FUNCTION "GetBitByte" : Bool   // FC2, SCL
{ S7_Optimized_Access := 'TRUE' }
VERSION : 0.1
   VAR_INPUT
      Data : Byte;
      pos : Int;
   END_VAR
   VAR_TEMP
      mask : Byte;
      temp : Byte;
   END_VAR
BEGIN
   #mask := 1;
   IF #pos < 8 THEN
       #mask := SHL(IN := #mask, N := #pos);
       #temp := #Data AND #mask;
       #GetBitByte := (#temp > 0);
   ELSE
       #GetBitByte := 0;
   END_IF;
END_FUNCTION

FUNCTION "GetBitWord" : Bool   // FC3, SCL
{ S7_Optimized_Access := 'TRUE' }
VERSION : 0.1
   VAR_INPUT
      Data : Word;
      pos : Int;
   END_VAR
   VAR_TEMP
      mask : Word;
      temp : Word;
   END_VAR
BEGIN
   #mask := 1;
   IF #pos < 16 THEN
       #mask := SHL(IN := #mask, N := #pos);
       #temp := #Data AND #mask;
       #GetBitWord := (#temp > 0);
   ELSE
       #GetBitWord := 0;
   END_IF;
END_FUNCTION

FUNCTION "SwapWord" : Void   // FC4, SCL
{ S7_Optimized_Access := 'TRUE' }
VERSION : 0.1
   VAR_INPUT
      NDB : Int;   // Номер DB-источника данных
      offset : Int;   // Смещение от начала DB, в байтах
      "counter" : Int;   // Число переворачиваемых WORD-ов
   END_VAR
   VAR_TEMP
      peek1 : Byte;
      peek2 : Byte;
      i : Int;
   END_VAR
BEGIN

   FOR #i := #offset TO #offset + (#counter - 1) * 2 BY 2 DO
       #peek1 := PEEK(area := 16#84,
                      dbNumber := #NDB,
                      byteOffset := #i);
       #peek2 := PEEK(area := 16#84,
                      dbNumber := #NDB,
                      byteOffset := #i + 1);
       POKE(area := 16#84,
            dbNumber := #NDB,
            byteOffset := #i + 1,
            value := #peek1);
       POKE(area := 16#84,
            dbNumber := #NDB,
            byteOffset := #i,
            value := #peek2);
   END_FOR;
END_FUNCTION

FUNCTION "Swap_float" : Void   // FC5, SCL
{ S7_Optimized_Access := 'TRUE' }
VERSION : 0.1
   VAR_INPUT
      offset : Int;
      "counter" : Int;
      NDB : Int;
   END_VAR
   VAR_TEMP
      i : Int;
      peek1 : Word;
      peek2 : Word;
   END_VAR
BEGIN
   FOR #i := #offset TO #offset + (#counter - 1) * 4 BY 4 DO
       #peek1 := PEEK_WORD(area := 16#84,
                           dbNumber := #NDB,
                           byteOffset := #i);
       #peek2 := PEEK_WORD(area := 16#84,
                           dbNumber := #NDB,
                           byteOffset := #i + 2);
       POKE(area := 16#84,
            dbNumber := #NDB,
            byteOffset := #i + 2,
            value := #peek1);
       POKE(area := 16#84,
            dbNumber := #NDB,
            byteOffset := #i,
            value := #peek2);
   END_FOR;
END_FUNCTION

FUNCTION "SetBitWord" : Void   // FC6, SCL
{ S7_Optimized_Access := 'TRUE' }
VERSION : 0.1
   VAR_INPUT
      pos : Int;
      value : Bool;
   END_VAR
   VAR_IN_OUT
      Data : Word;
   END_VAR
   VAR_TEMP
      mask : Word;
      v : Word;
   END_VAR
BEGIN
   IF #pos < 16 THEN
       #mask := 1;
       #mask := SHL(IN := #mask, N := #pos);
       IF #value THEN
           #Data := #Data OR #mask;
       ELSE
           #Data := #Data AND (NOT #mask);
       END_IF;
   END_IF;
END_FUNCTION

FUNCTION "SetBitByte" : Void   // FC7, SCL
{ S7_Optimized_Access := 'TRUE' }
VERSION : 0.1
   VAR_INPUT
      pos : Int;
      value : Bool;
   END_VAR
   VAR_IN_OUT
      Data : Byte;
   END_VAR
   VAR_TEMP
      mask : Byte;
      v : Byte;
   END_VAR
BEGIN
   IF #pos < 8 THEN
       #mask := 1;
       #mask := SHL(IN := #mask, N := #pos);
       IF #value THEN
           #Data := #Data OR #mask;
       ELSE
           #Data := #Data AND (NOT #mask);
       END_IF;
   END_IF;
END_FUNCTION

// folder: Modbus

FUNCTION "UVP_Processing" : Void   // FC9, SCL
{ S7_Optimized_Access := 'TRUE' }
VERSION : 0.1
   VAR_TEMP
      NewState : Int;
      Cant_connect1 : Bool;
      Cant_connect2 : Bool;
      Cant_connect_with_UVP : Bool;
      Request_Finished : Bool;
      Request_Finished_with_Error : Bool;
      len : UInt;
   END_VAR
BEGIN
   // Установить IP адрес УВП
   (*IF "UVP_Data".Commands.Set_IP_UVP1 THEN
       IF NOT "UVP_States".Client.Disconnect THEN
           "UVP_States".Connect_UVP.ID := UINT_TO_WORD("UVP_Data".UVP1_Settings.Connect_ID);
           "UVP_States".Connect_UVP.RemoteAddress.ADDR[1] := UINT_TO_BYTE("UVP_Data".UVP1_Settings.IP_OCTET1);
           "UVP_States".Connect_UVP.RemoteAddress.ADDR[2] := UINT_TO_BYTE("UVP_Data".UVP1_Settings.IP_OCTET2);
           "UVP_States".Connect_UVP.RemoteAddress.ADDR[3] := UINT_TO_BYTE("UVP_Data".UVP1_Settings.IP_OCTET3);
           "UVP_States".Connect_UVP.RemoteAddress.ADDR[4] := UINT_TO_BYTE("UVP_Data".UVP1_Settings.IP_OCTET4);
           "UVP_States".Connect_UVP.RemotePort := "UVP_Data".UVP1_Settings.IP_PORT;
           "UVP_States".State := 10;
           "UVP_States".Client.Disconnect := True;
       ELSE
           "UVP_States".Client.Disconnect := False;
           "UVP_Data".Commands.Set_IP_UVP1 := False;
       END_IF;
   END_IF;*)

   #NewState := -1;

   // определение проблем с подключением
   #Request_Finished := "UVP_States".Client.Done OR "UVP_States".Client.Error OR ("UVP_States".Client.Busy AND ("UVP_States".Client.Status = 16#7002));
   // признак завершения цикла работы чтения/записи с ошибкой
   #Request_Finished_with_Error := ("UVP_States".Client.Busy AND ("UVP_States".Client.Status = 16#7002)) OR
   ("UVP_States".Client.Error AND (("UVP_States".Client.Status <> 16#7002)));

   // определение проблем со связью
   IF ("UVP_States".Client.Busy OR "UVP_States".Client.Error) THEN
       "UVP_off".TON (IN := true, PT := t#5s);
       IF "UVP_off".Q THEN
           "UVP_Data".Flags.UVP1_on := false;
           "ReqUVP" := 0;
           #NewState := "UVP_States".ReqReadOpData_nextState;
           "UVP_off".TON (IN := false, PT := t#5s);
       END_IF;
   ELSE
       "UVP_off".TON (IN := false, PT := t#5s);
   END_IF;

   IF "UVP_States".Client.Done AND (NOT "UVP_States".Client.Error) THEN
       "UVP_Data".Flags.UVP1_on := true;
   END_IF;

   (*IF "ReqUVP" THEN
       "ReqUVP" := 0;
   ELSE
       IF NOT ("UVP_States".Client.Done OR "UVP_States".Client.Error OR "UVP_States".Client.Busy) THEN
           "ReqUVP" := 1;
       END_IF;
   END_IF;*)


   CASE "UVP_States".State OF
       10..29:// State=10 - чтение оперативных данных первой линии, параметры с 3 по 23
           // State=11 - чтение накопленных данных первой линии, 4 группы по 5 параметров
           // State=12 - чтение оперативных данных первой линии, параметры с 1 по 3
           // 
           // State=13 - чтение оперативных данных второй линии, параметры с 3 по 23
           // State=14 - чтение накопленных данных второй линии, 4 группы по 5 параметров
           // State=15 - чтение оперативных данных второй линии, параметры с 1 по 3

           // 
           IF ("PrevState" <> "UVP_States".State) THEN
               "UVP_States".ReqReadOpData.Mode := 0;
               //ил 1
               IF "UVP_States".State = 10 THEN
                   "UVP_States".ReqReadOpData.Data_ADDR := 32001;
                   "UVP_States".ReqReadOpData.Data_LEN := 46;
                   "UVP_States".ReqReadOpData_dest_offset := 64; // смещение проверить в Дата
                   "UVP_States".ReqReadOpData_nextState := 11;
               ELSIF "UVP_States".State = 11 THEN
                   "UVP_States".ReqReadOpData.Data_ADDR := 32061;
                   "UVP_States".ReqReadOpData.Data_LEN := 40;
                   "UVP_States".ReqReadOpData_dest_offset := 156; // смещение проверить в Дата
                   "UVP_States".ReqReadOpData_nextState := 13;

                   //ил 2    
               ELSIF "UVP_States".State = 13 THEN
                   "UVP_States".ReqReadOpData.Data_ADDR := 32101;
                   "UVP_States".ReqReadOpData.Data_LEN := 46;
                   "UVP_States".ReqReadOpData_dest_offset := 236;
                   "UVP_States".ReqReadOpData_nextState := 14;
               ELSIF "UVP_States".State = 14 THEN
                   "UVP_States".ReqReadOpData.Data_ADDR := 32161;
                   "UVP_States".ReqReadOpData.Data_LEN := 40;
                   "UVP_States".ReqReadOpData_dest_offset := 328;
                   "UVP_States".ReqReadOpData_nextState := 30;
               END_IF;
               "ReqUVP" := 0;
               "UVP_States".ClientMode := "UVP_States".ReqReadOpData;
               "ReqUVP" := 1;

           END_IF;
           // обработка принятых данных
           IF "UVP_States".Client.Done THEN
               // перекладываем прочитаные данные в секцию UVP_Current_L1(L2), UVP_Current_L1(L2)  или UVP_Cumulative_L1(L3), смотря по запросу              
               "CopyWord"(NDBsrc := 14,
                          NDBdest := 13,
                          offset_src := 52,
                          offset_dest := "UVP_States".ReqReadOpData_dest_offset,
                          counter := UINT_TO_INT("UVP_States".ReqReadOpData.Data_LEN));
               "ReqUVP" := 0;
               // постобработка данных - перевожу Па в МПа, секундные расходы в часовые
               IF "UVP_States".State = 10 THEN
                   "UVP_Data".UVP1_Current_L1.UVP_mass_flow := "UVP_Data".UVP1_Current_L1.UVP_mass_flow * 3600.0;
                   "UVP_Data".UVP1_Current_L1.UVP_Param_m_flow := "UVP_Data".UVP1_Current_L1.UVP_Param_m_flow * 3600.0;
                   "UVP_Data".UVP1_Current_L1.UVP_Param_vol_flow_norm := "UVP_Data".UVP1_Current_L1.UVP_Param_vol_flow_norm * 3600.0;
                   "UVP_Data".UVP1_Current_L1.UVP_Param_vol_flow_work := "UVP_Data".UVP1_Current_L1.UVP_Param_vol_flow_work * 3600.0;
                   "UVP_Data".UVP1_Current_L1.UVP_vol_flow_norm := "UVP_Data".UVP1_Current_L1.UVP_vol_flow_norm * 3600.0;
                   "UVP_Data".UVP1_Current_L1.UVP_vol_flow_work := "UVP_Data".UVP1_Current_L1.UVP_vol_flow_work * 3600.0;
                   "UVP_Data".UVP1_Current_L1.UVP_Abs_press := "UVP_Data".UVP1_Current_L1.UVP_Abs_press / 1000000;
                   "UVP_Data".UVP1_Current_L1.UVP_Press := "UVP_Data".UVP1_Current_L1.UVP_Press / 1000000;
               ELSIF "UVP_States".State = 11 THEN
                   "UVP_Data".UVP1_Cumulative_L1.UVP_Mass_prev2h := "UVP_Data".UVP1_Cumulative_L1.UVP_Mass_prev2h / 1000.0;
                   "UVP_Data".UVP1_Cumulative_L1.UVP_Param_m_flow_prev2h := "UVP_Data".UVP1_Cumulative_L1.UVP_Param_m_flow_prev2h / 1000.0;
                   "UVP_Data".UVP1_Cumulative_L1.UVP_Mass_prevDay := "UVP_Data".UVP1_Cumulative_L1.UVP_Mass_prevDay / 1000.0;
                   "UVP_Data".UVP1_Cumulative_L1.UVP_Param_m_flow_prevDay := "UVP_Data".UVP1_Cumulative_L1.UVP_Param_m_flow_prevDay / 1000.0;
               ELSIF "UVP_States".State = 13 THEN
                   "UVP_Data".UVP1_Current_L2.UVP_mass_flow := "UVP_Data".UVP1_Current_L2.UVP_mass_flow * 3.6;
                   "UVP_Data".UVP1_Current_L2.UVP_Param_m_flow := "UVP_Data".UVP1_Current_L2.UVP_Param_m_flow * 3600.0;
                   "UVP_Data".UVP1_Current_L2.UVP_Param_vol_flow_norm := "UVP_Data".UVP1_Current_L2.UVP_Param_vol_flow_norm * 3600.0;
                   "UVP_Data".UVP1_Current_L2.UVP_Param_vol_flow_work := "UVP_Data".UVP1_Current_L2.UVP_Param_vol_flow_work * 3600.0;
                   "UVP_Data".UVP1_Current_L2.UVP_vol_flow_norm := "UVP_Data".UVP1_Current_L2.UVP_vol_flow_norm * 3600.0;
                   "UVP_Data".UVP1_Current_L2.UVP_vol_flow_work := "UVP_Data".UVP1_Current_L2.UVP_vol_flow_work * 3600.0;
                   "UVP_Data".UVP1_Current_L2.UVP_Abs_press := "UVP_Data".UVP1_Current_L2.UVP_Abs_press / 1000000;
                   "UVP_Data".UVP1_Current_L2.UVP_Press := "UVP_Data".UVP1_Current_L2.UVP_Press / 1000000;
               ELSIF "UVP_States".State = 14 THEN
                   "UVP_Data".UVP1_Cumulative_L2.UVP_Mass_prev2h := "UVP_Data".UVP1_Cumulative_L2.UVP_Mass_prev2h / 1000.0;
                   "UVP_Data".UVP1_Cumulative_L2.UVP_Param_m_flow_prev2h := "UVP_Data".UVP1_Cumulative_L2.UVP_Param_m_flow_prev2h / 1000.0;
                   "UVP_Data".UVP1_Cumulative_L2.UVP_Mass_prevDay := "UVP_Data".UVP1_Cumulative_L2.UVP_Mass_prevDay / 1000.0;
                   "UVP_Data".UVP1_Cumulative_L2.UVP_Param_m_flow_prevDay := "UVP_Data".UVP1_Cumulative_L2.UVP_Param_m_flow_prevDay / 1000.0;
               END_IF;
               // Переходим к следующему запросу
               #NewState := "UVP_States".ReqReadOpData_nextState;
           ELSIF #Request_Finished_with_Error THEN
               // Если не получается связаться - переходим к следующему запросу и продолжаем попытки
               #NewState := "UVP_States".ReqReadOpData_nextState;
           ELSE
               ;
           END_IF;

           //******************** проверка команд*************************************************************************************************

           IF "UVP_Data".Commands.UVPArchReadStart THEN
               // переход к чтению архивной записи
               #NewState := 55;
               //ELSIF "UVP_Data".Commands.UVP_MR113_Read THEN         //читаем циклически
               // переход к чтению компонентного состава газа
               //    #NewState := 40;
           ELSIF "UVP_Data".Commands.UVP_MR113_Write THEN
               // переход к записи компонентного состава газа
               #NewState := 50;

           ELSE
               // нет команды
               ;
           END_IF;

       30:  //  чтение часов реального времени выбранного УВП, сразу после измеряемых параметров УВП по обоим линиям         
           IF NOT "UVP_States".Client.Busy THEN
               "UVP_States".ReqReadOpData.Mode := 0;
               "UVP_States".ReqReadOpData.Data_ADDR := 41801;
               "UVP_States".ReqReadOpData.Data_LEN := 6;
               "ReqUVP" := 0;
               "UVP_States".ClientMode := "UVP_States".ReqReadOpData;
               "ReqUVP" := 1;
               #NewState := 31;
           END_IF;

       31: // обработка принятых данных часов реального времени выбранного УВП
           // крутить их не нужно, так как в УВП они в нормальном представлении
           IF "UVP_States".Client.Done THEN
               // перекладываем прочитаные данные в секцию UVP_DateTime
               "CopyWord"(NDBsrc := 14,
                          NDBdest := 13,
                          offset_src := 52,
                          offset_dest := 924,
                          counter := 6);
               "ReqUVP" := 0;
               #NewState := 32;
           ELSIF #Request_Finished_with_Error THEN
               // Если не получается связаться - переходим к следующему запросу и продолжаем попытки
               #NewState := 32;
           ELSE
               ;
           END_IF;

       32:  //  запись нужного порядка байт в 4-х байтной переменной         
           IF NOT "UVP_States".Client.Busy THEN
               "UVP_States".ReqWriteCom.Mode := 1;
               "UVP_States".ReqWriteCom.Data_ADDR := 40101;
               "UVP_States".ReqWriteCom.Data_LEN := 1;
               "ReqUVP" := 0;
               %DB14.DBW52 := 291;                                  // это 0123h
               "UVP_States".ClientMode := "UVP_States".ReqWriteCom;
               "ReqUVP" := 1;
               #NewState := 33;
           END_IF;

       33: // ожидание завершения записи порядка байт
           IF #Request_Finished THEN
               // Возвращаемся к очередному запросу (с которого нас сняли командой)
               #NewState := 40;
               "ReqUVP" := 0;
           END_IF;


       40:  // State=40 - запуск чтения компонентного состава газа
           IF NOT "UVP_States".Client.Busy THEN
               "UVP_States".ReqReadOpData.Mode := 0;
               "UVP_States".ReqReadOpData.Data_ADDR := 41103;
               "UVP_States".ReqReadOpData.Data_LEN := 30;
               "ReqUVP" := 0;
               "UVP_States".ClientMode := "UVP_States".ReqReadOpData;
               "ReqUVP" := 1;
               #NewState := 41;
           END_IF;

       41: // State=41 - обработка принятых данных компонентного состава газа
           IF "UVP_States".Client.Done THEN
               // перекладываем прочитаные данные в секцию UVP_MR113
               "CopyWord"(NDBsrc := 14,
                          NDBdest := 13,
                          offset_src := 52,
                          offset_dest := 936,
                          counter := 30);
               "ReqUVP" := 0;
               // Возвращаемся к очередному запросу (с которого нас сняли командой)
               #NewState := 42;
               "UVP_Data".Commands.UVP_MR113_Read := False;
           ELSIF #Request_Finished_with_Error THEN
               // Если не получается связаться - переходим к следующему запросу и продолжаем попытки
               #NewState := 42;
               //"UVP_v2_Data".Commands.UVP_MR113_Read := False; // Из-за этого не читает комп. состав при загрузке контроллера
           ELSE
               ;
           END_IF;


       42:  // State=42 - запуск чтения параметров: молярная или массовая концентрация,  влажность
           IF NOT "UVP_States".Client.Busy THEN
               "UVP_States".ReqReadOpData.Mode := 0;
               "UVP_States".ReqReadOpData.Data_ADDR := 41101;
               "UVP_States".ReqReadOpData.Data_LEN := 2;
               "ReqUVP" := 0;
               "UVP_States".ClientMode := "UVP_States".ReqReadOpData;
               "ReqUVP" := 1;
               #NewState := 43;
           END_IF;

       43: // State=43 - обработка принятых параметров: молярная или массовая концентрация,  влажность
           IF "UVP_States".Client.Done THEN
               // перекладываем прочитаные данные в секцию UVP_MR113
               // крутить их не нужно, так как в УВП они в нормальном представлении
               "CopyWord"(NDBsrc := 14,
                          NDBdest := 13,
                          offset_src := 52,
                          offset_dest := 996,
                          counter := 2);
               "ReqUVP" := 0;
               // Возвращаемся к очередному запросу (с которого нас сняли командой)
               #NewState := 10;
           ELSIF #Request_Finished_with_Error THEN
               // Если не получается связаться - переходим к следующему запросу и продолжаем попытки
               #NewState := 10;
           ELSE
               ;
           END_IF;// конец            

       50:  // State=50 - запись компонентного состава газа
           IF NOT "UVP_States".Client.Busy THEN
               "UVP_States".ReqWriteCom.Mode := 1;
               "UVP_States".ReqWriteCom.Data_ADDR := 41103;
               "UVP_States".ReqWriteCom.Data_LEN := 30;
               "ReqUVP" := 0;
               "CopyWord"(NDBsrc := 57,
                          NDBdest := 33,
                          offset_src := 1740,
                          offset_dest := 86,
                          counter := 30);
               "UVP_States".ClientMode := "UVP_States".ReqWriteCom;
               "ReqUVP" := 1;
               #NewState := 52;
               "UVP_Data".Commands.UVP_MR113_Write := False;
           END_IF;

       52:  // ожидание завершения записи компонентного состава газа
           IF #Request_Finished THEN
               // Возвращаемся к очередному запросу (с которого нас сняли командой)
               #NewState := 53;
           END_IF;

       53:  // State=53 - запись параметров: молярная или массовая концентрация,  влажность
           IF NOT "UVP_States".Client.Busy THEN
               "UVP_States".ReqWriteCom.Mode := 1;
               "UVP_States".ReqWriteCom.Data_ADDR := 41101;
               "UVP_States".ReqWriteCom.Data_LEN := 2;
               "ReqUVP" := 0;
               // крутить их не нужно, так как в УВП они в нормальном представлении        
               "CopyWord"(NDBsrc := 57,
                          NDBdest := 33,
                          offset_src := 1800,
                          offset_dest := 86,
                          counter := 2);
               "UVP_States".ClientMode := "UVP_States".ReqWriteCom;
               "ReqUVP" := 1;
               #NewState := 54;
               "UVP_Data".Commands.UVP_MR113_Write := False;
           END_IF;

       54:  // ожидание завершения записи молярной или массовой концентрации,  влажности
           IF #Request_Finished THEN
               // Возвращаемся к очередному запросу (с которого нас сняли командой)
               #NewState := "UVP_States".ReqReadOpData_nextState;
           END_IF;

           //---------------------------------------------------------------------------------------------------------------------               
           //------------------------------ АРХИВЫ -------------------------------------------------------------------------------         
           (*           
           55:  // - запись параметров запроса на чтение архивных данных
               IF NOT "UVP2_States".Client.Busy THEN
                   "UVP2_States".ReqWriteCom.Mode := 1;
                   "UVP2_States".ReqWriteCom.Data_ADDR := 47901;
                   "UVP2_States".ReqWriteCom.Data_LEN := 14;
                   "Req2" := 0;
                       "CopyWord"(NDBsrc := 57,
                                  NDBdest := 33,
                                  offset_src := 1804,
                                  offset_dest := 86,
                                  counter := 14);

                   // Так как для УВП год вводится в формате "Число лет с 2000 г", а пользователю удобнее вводить полный год,
                   // принимаем год в обычном формате, а в УВП пишем число на 2000 меньше
                   // "UVP2_States".Data_PTR[4]  := "UVP2_States".Data_PTR[4]  - 2000;
                   // "UVP2_States".Data_PTR[10] := "UVP2_States".Data_PTR[10] - 2000;
                   "UVP2_States".ClientMode := "UVP2_States".ReqWriteCom;
                   "Req2" := 1;
                   #NewState := 56;

               END_IF;

           56:  //  - ожидание записи параметров запроса на чтение архива в УВП, переход в режим записи формата запроса
               IF "UVP2_States".Client.Done THEN
                   #NewState := 57;
               ELSIF #Request_Finished_with_Error THEN
                   #NewState := "UVP2_States".ReqReadOpData_nextState;
               ELSE
                   ;
               END_IF;

           57: //  - запись формата запроса архивных данных (по нему стартует формирование архива в УВП)
               "UVP2_States".ReqWriteCom.Mode := 1;
               "UVP2_States".ReqWriteCom.Data_ADDR := 47915;
               "UVP2_States".ReqWriteCom.Data_LEN := 1;
               "Req2" := 0;
               "UVP2_States".Data_PTR[0] := "UVP2_States".Format;
               "UVP2_States".ClientMode := "UVP2_States".ReqWriteCom;
               "Req2" := 1;
               // Можно начинать ждать архивных данных
               #NewState := 58;

           58: // - ожидание записи формата запроса       
               IF "UVP2_States".Client.Done THEN
                   #NewState := 59;
               ELSIF #Request_Finished_with_Error THEN
                   #NewState := "UVP2_States".ReqReadOpData_nextState;
               ELSE
                   ;
               END_IF;

           59://  - чтение состояния готовности данных
               "UVP_Data".UVP2_Flags.RezNonValid := 0;
               "UVP_Data".UVP2_Flags.NonNote := 0;
               "UVP_Data".UVP2_Flags.NonCorPrimDate := 0;
               "UVP_Data".UVP2_Flags.NonCorFinDate := 0;
               "UVP_Data".UVP2_Flags.NonCorNumLine := 0;
               "UVP_Data".UVP2_Flags.LargePeriod := 0;
               // чтение состояния готовности данных
               "UVP2_States".ReqReadAns.Mode := 0;
               "UVP2_States".ReqReadAns.Data_ADDR := 48001;
               "UVP2_States".ReqReadAns.Data_LEN := 2;
               "Req2" := 0;
               "UVP2_States".ClientMode := "UVP2_States".ReqReadAns;
               "Req2" := 1;
               // обработка состояния готовности
               IF "UVP2_States".Client.Done THEN
                   "UVP2_States".Answer := "UVP2_States".Data_PTR[0];
                   // статус запроса архива УВП обновляем отсюда
                       "UVP_Data".Archive_Results.UVP2_Archive_RequestStatus := WORD_TO_INT("UVP2_States".Data_PTR[0]);
                       "UVP_Data".Archive_Results.UVP2_Archive_Update_Data := WORD_TO_INT("UVP2_States".Data_PTR[1]);

                   // данные готовы - переходим к их парсингу
                   IF "UVP2_States".Answer = 16#0002 THEN
                       #NewState := 60;
                   ELSE
                       // результат запроса уничтожен по таймауту или запрос не был воспринят вычислителем
                       IF "UVP2_States".Answer = 16#0000 THEN
                           "UVP_Data".Flags.RezNonValid := 1;
                           #NewState := 10;
                       END_IF;
                       // за выбранный промежуток времени в архиве нет ни одной записи  
                       IF "UVP2_States".Answer = 16#0003 THEN
                           "UVP_Data".Flags.NonNote := 1;
                           #NewState := 10;
                       END_IF;
                       // ошибка в начальном времени, дата или время некорректны
                       IF "UVP2_States".Answer = 16#0004 THEN
                           "UVP_Data".Flags.NonCorPrimDate := 1;
                           #NewState := 10;
                       END_IF;
                       // ошибка в конечном времени, дата или время некорректны
                       IF "UVP2_States".Answer = 16#0005 THEN
                           "UVP_Data".Flags.NonCorFinDate := 1;
                           #NewState := 10;
                       END_IF;
                       // ошибка в задании номера трубопровода
                       IF "UVP2_States".Answer = 16#0006 THEN
                           "UVP_Data".Flags.NonCorNumLine := 1;
                           #NewState := 10;
                       END_IF;
                       // выбран слишком большой период для сбора данных, сбор данных продолжался больше 15 секунд
                       IF "UVP2_States".Answer = 16#0007 THEN
                           "UVP_Data".Flags.LargePeriod := 1;
                           #NewState := 10;
                       END_IF;
                       // остаётся вариант "UVP2_States".Answer = 16#0001 - идет сбор данных. По нему достаточно ждать 
                   END_IF;
               ELSIF #Request_Finished_with_Error THEN
                   #NewState := "UVP2_States".ReqReadOpData_nextState;
               ELSE
                   ;
               END_IF;
           60: //  - запрашиваем строку архива
               IF NOT "UVP2_States".Client.Busy THEN
                   "UVP2_States".ReqReadArcData.Mode := 0;
                   "UVP2_States".ReqReadArcData.Data_ADDR := 48003;
                   "UVP2_States".ReqReadArcData.Data_LEN := 120;
                   "Req2" := 0;
                   "UVP2_States".ClientMode := "UVP2_States".ReqReadArcData;
                   "Req2" := 1;
                   #NewState := 61;
               END_IF;

           61: // - обработка полученой строки архива
               IF "UVP2_States".Client.Done THEN
                   "CopyWord"(NDBsrc := 33,
                              NDBdest := 58,
                              offset_src := 86,
                              offset_dest := 0,
                              counter := 120);

                   #len := CHAR_TO_UINT("ArcDataDB_UVP2".ArcData[1]) + (CHAR_TO_UINT("ArcDataDB_UVP2".ArcData[0]) * 256) - 1;
                   Chars_TO_Strg(Chars := "ArcDataDB_UVP2".ArcData,
                                 pChars := 2,
                                 Cnt := #len,
                                 Strg => "UVP2_States".ArcDataString);
                   // данные кладём в нужную линию сразу
                   "ParseString_2"(ClientIndex := 1);

                   #NewState := "UVP2_States".ReqReadOpData_nextState;

               ELSIF #Request_Finished_with_Error THEN
                   #NewState := "UVP2_States".ReqReadOpData_nextState;
               ELSE
                   ;
               END_IF;
    *)
    // Если случайно State кривой - начнём с начала
   ELSE
       #NewState := 10;
   END_CASE;

   "PrevState" := "UVP_States".State;

   IF #NewState >= 0 THEN
       "UVP_States".State := #NewState;
   END_IF;
END_FUNCTION

FUNCTION "REG_Processing" : Void   // FC10, SCL
{ S7_Optimized_Access := 'FALSE' }
VERSION : 0.1
   VAR_TEMP
      Request_Finished : Bool;
      Request_Finished_with_Error : Bool;
   END_VAR
BEGIN
   // Если порт не поднят, поднимаем
   IF NOT "Modbus_Comm_Load_Regs".DONE THEN
       "Modbus_Comm_Load_Regs".MODE := 4; // Operating mode 4 = Half duplex (RS485) two-wire mode
       "Modbus_Comm_Load_Regs"(REQ := true,
                               "PORT" := "PortSettings".Regs."Port",
                               BAUD := "PortSettings".Regs.Baud,
                               PARITY := "PortSettings".Regs.Parity,
                               FLOW_CTRL := 0,
                               RTS_ON_DLY := 0,
                               RTS_OFF_DLY := 0,
                               RESP_TO := 1000,
                               DONE => "PortSettings".Regs.Done,
                               ERROR => "PortSettings".Regs.Error,
                               STATUS => "PortSettings".Regs.Status,
                               MB_DB := "Modbus_Master_Regs".MB_DB);
   END_IF;

   // *********************************************Диагностика ошибок**********************************************************
   #Request_Finished := "REG_Master".Settings.Done OR "REG_Master".Settings.Error;
   // признак завершения цикла работы чтения/записи с ошибкой
   #Request_Finished_with_Error :=
   "REG_Master".Settings.Error AND ((("REG_Master".Settings.Status = 16#8380)) OR (("REG_Master".Settings.Status = 16#8381)) OR (("REG_Master".Settings.Status = 16#8382)) OR (("REG_Master".Settings.Status = 16#8383)) OR (("REG_Master".Settings.Status = 16#8384)) OR (("REG_Master".Settings.Status = 16#8385)) OR (("REG_Master".Settings.Status = 16#8386)) OR (("REG_Master".Settings.Status = 16#8387)) OR (("REG_Master".Settings.Status = 16#8388)));

   // блок обработки ошибки связи
   IF (("REG_Master".Settings.Status <> 16#0000) AND ("REG_Master".Settings.Status <> 16#7000) AND ("REG_Master".Settings.Status <> 16#7001) AND ("REG_Master".Settings.Status <> 16#7002)) THEN
       IF "REG_Master".Settings.MB_Addr = 1 THEN
           "REG_Master".PCV300_error := TRUE;
       END_IF;
       IF "REG_Master".Settings.MB_Addr = 2 THEN
           "REG_Master".LCV300_error := TRUE;
       END_IF;
   END_IF;

   // блок сброса ошибки связи
   IF "REG_Master".Settings.Done AND (NOT "REG_Master".Settings.Error) THEN
       IF "REG_Master".Settings.MB_Addr = 1 THEN
           "REG_Master".PCV300_error := false;
       END_IF;
       IF "REG_Master".Settings.MB_Addr = 2 THEN
           "REG_Master".LCV300_error := false;
       END_IF;
   END_IF;

   //*********************************************************************************************

   // 10 - чтение с регулятора PCV300, сетевой адрес 1
   // 11 - чтение с регулятора LCV300, сетевой адрес 2 
   // 13 - запись в PCV300 задания положения
   // 14 - запись в LCV300 задания положения 

   IF "REG_Master".State = 10 THEN

       IF "REG_Master".State = 10 AND "REG_Master".reg_PCV300_err = true THEN
           IF "REG_Master".count_PCV300 < 1000 THEN
               "REG_Master".State := 11;
               "REG_Master".count_PCV300 := "REG_Master".count_PCV300 + 1;
           ELSIF "REG_Master".count_PCV300 >= 1000 THEN
               "REG_Master".count_PCV300 := 0;
               "REG_Master".reg_PCV300_err := false;
           END_IF;
       END_IF;

       IF "REG_Master".State = 10 AND "REG_Master".reg_PCV300_err = false THEN
           "REG_Master".MasterMode.Mode := 0;
           "REG_Master".Settings.MB_Addr := 1;
           "REG_Master".MasterMode.Data_Addr := 31001;
           "REG_Master".MasterMode.Data_Len := 3;
           "REG_Master".Data_offset := 2;
           "REG_Master".Register := 3;
           "REG_Master".Next_State := 11;
           "REG_Master".reqREGmaster := 1;
       END_IF;
   END_IF;

   IF "REG_Master".State = 11 THEN
       IF "REG_Master".State = 11 AND "REG_Master".reg_LCV300_err = true THEN
           IF "REG_Master".count_LCV300 < 1000 THEN
               "REG_Master".State := 13;
               "REG_Master".count_LCV300 := "REG_Master".count_LCV300 + 1;
           ELSIF "REG_Master".count_LCV300 >= 1000 THEN
               "REG_Master".count_LCV300 := 0;
               "REG_Master".reg_LCV300_err := false;
           END_IF;
       END_IF;

       IF "REG_Master".State = 11 AND "REG_Master".reg_LCV300_err = false THEN
           "REG_Master".MasterMode.Mode := 0;
           "REG_Master".Settings.MB_Addr := 2;
           "REG_Master".MasterMode.Data_Addr := 31001;
           "REG_Master".MasterMode.Data_Len := 3;
           "REG_Master".Data_offset := 14;
           "REG_Master".Register := 3;
           "REG_Master".Next_State := 13;
           "REG_Master".reqREGmaster := 1;
       END_IF;
   END_IF;

   IF "REG_Master".State = 13 THEN
       // переходим на запись положений (SP)

       IF "REG_Master".State = 13 AND "REG_Master".reg_PCV300_err = true THEN
           "REG_Master".State := 14;
       END_IF;

       IF "REG_Master".State = 13 AND "REG_Master".reg_PCV300_err = false THEN
           "REG_Master".MasterMode.Mode := 1;
           "REG_Master".Settings.MB_Addr := 1;
           "REG_Master".MasterMode.Data_Addr := 41001;
           "REG_Master".MasterMode.Data_Len := 2;
           "REG_Master".Register := 1;
           "REG_Master".Next_State := 14;
           %DB16.DBW6 := 1024;
           "CopyWord"(NDBsrc := 15,
                      NDBdest := 16,
                      offset_src := 12,
                      offset_dest := 8,
                      counter := "REG_Master".Register);
           "REG_Master".reqREGmaster := 1;
       END_IF;
   END_IF;

   IF "REG_Master".State = 14 THEN
       IF "REG_Master".State = 14 AND "REG_Master".reg_LCV300_err = true THEN
           "REG_Master".State := 10;
       END_IF;

       IF "REG_Master".State = 14 AND "REG_Master".reg_LCV300_err = false THEN
           "REG_Master".MasterMode.Mode := 1;
           "REG_Master".Settings.MB_Addr := 2;
           "REG_Master".MasterMode.Data_Addr := 41001;
           "REG_Master".MasterMode.Data_Len := 2;
           "REG_Master".Register := 1;
           "REG_Master".Next_State := 10;
           %DB16.DBW6 := 1024;
           "CopyWord"(NDBsrc := 15,
                      NDBdest := 16,
                      offset_src := 24,
                      offset_dest := 8,
                      counter := "REG_Master".Register);
           "REG_Master".reqREGmaster := 1;
       END_IF;
   END_IF;

   IF "REG_Master".State = 10 OR "REG_Master".State = 11 OR "REG_Master".State = 12 THEN

       // обработка принятых данных
       IF "REG_Master".Settings.Done THEN
           IF "REG_Master".reg_PCV300_err = false OR "REG_Master".reg_LCV300_err = false THEN
               //"SwapWord"(NDB := 57,
               //           offset := 6,
               //           counter := 1);
               //"SwapWord"(NDB := 57,
               //           offset := 10,
               //           counter := 1);
               "CopyWord"(NDBsrc := 16,//пересылка из буфера в DBшку
                          NDBdest := 15,
                          offset_src := 6,
                          offset_dest := "REG_Master".Data_offset,
                          counter := "REG_Master".Register);

               IF ("REG_Master".State = 10) THEN
                   "REG_Master".PCV300_done_count := "REG_Master".PCV300_done_count + 1;
                   "REG_Master".PCV300_error := false;
                   IF ("REG_Master".PCV300_done_count >= 10000) THEN
                       "REG_Master".PCV300_done_count := 0;
                   END_IF;
               ELSIF ("REG_Master".State = 11) THEN
                   "REG_Master".LCV300_done_count := "REG_Master".LCV300_done_count + 1;
                   "REG_Master".LCV300_error := false;
                   IF ("REG_Master".LCV300_done_count >= 10000) THEN
                       "REG_Master".LCV300_done_count := 0;
                   END_IF;
               END_IF;

               IF NOT "REG_Master".Settings.Busy THEN
                   "REG_Master".State := "REG_Master".Next_State;
                   "REG_Master".reqREGmaster := 0;
               END_IF;
           ELSIF #Request_Finished_with_Error THEN
               "REG_Master".State := "REG_Master".Next_State;
               "REG_Master".reqREGmaster := 0;
           END_IF;
       END_IF;

       IF "REG_Master".State = 10 OR "REG_Master".State = 11 OR "REG_Master".State = 12 THEN
           IF ("REG_Master".Settings.Busy OR "REG_Master".Settings.Error) THEN
               "Timer_Busy_Modbus_Reg".TON(IN := true, PT := t#5s);
               IF "Timer_Busy_Modbus_Reg".Q THEN

                   IF "REG_Master".State = 10 THEN
                       "REG_Master".reg_PCV300_err := true;
                       "REG_Master".count_PCV300 := 0;
                       "REG_Master".PCV300_error := true;
                   END_IF;

                   IF "REG_Master".State = 11 THEN
                       "REG_Master".reg_LCV300_err := true;
                       "REG_Master".count_LCV300 := 0;
                       "REG_Master".LCV300_error := true;
                   END_IF;

                   "REG_Master".reqREGmaster := 0;
                   "REG_Master".State := "REG_Master".Next_State;
                   "Timer_Busy_Modbus_Reg".TON(IN := false, PT := t#5s);
               END_IF;
           ELSE
               "Timer_Busy_Modbus_Reg".TON(IN := false, PT := t#5s);
           END_IF;
       END_IF;

   END_IF;


   IF "REG_Master".State = 13 OR "REG_Master".State = 14 OR "REG_Master".State = 15 THEN

       //"REG_Master".MasterMode.Mode := 1;

       IF "REG_Master".Settings.Done THEN
           IF "REG_Master".State = 13 OR "REG_Master".State = 14 OR "REG_Master".State = 15 THEN
               IF NOT "REG_Master".Settings.Busy THEN
                   "REG_Master".State := "REG_Master".Next_State;
                   "REG_Master".reqREGmaster := 0;
               ELSIF #Request_Finished_with_Error THEN
                   "REG_Master".State := "REG_Master".Next_State;
                   "REG_Master".reqREGmaster := 0;
               END_IF;
           END_IF;
       END_IF;

       IF ("REG_Master".Settings.Busy OR "REG_Master".Settings.Error) THEN
           "Timer_Busy_Modbus_Reg2".TON(IN := true, PT := t#5s);
           IF "Timer_Busy_Modbus_Reg2".Q THEN

               //-----На случай если данные прочитались с регулятора, но не записались--------------
               IF "REG_Master".State = 13 THEN
                   "REG_Master".reg_PCV300_err := true;
                   "REG_Master".count_PCV300 := 0;
                   "REG_Master".PCV300_error := true;
               END_IF;

               IF "REG_Master".State = 14 THEN
                   "REG_Master".reg_LCV300_err := true;
                   "REG_Master".count_LCV300 := 0;
                   "REG_Master".LCV300_error := true;
               END_IF;

               //----------------------------------------------------------------------------------

               "REG_Master".reqREGmaster := 0;
               "REG_Master".State := "REG_Master".Next_State;
               "Timer_Busy_Modbus_Reg2".TON(IN := false, PT := t#5s);
           END_IF;
       ELSE
           "Timer_Busy_Modbus_Reg2".TON(IN := false, PT := t#5s);
       END_IF;
   END_IF;


   // приведение положения регулятора с 100% шкале

   "REG_Data".PCV300_Pologenie_ok := INT_TO_REAL("REG_Data".PCV300_Pologenie) / 10;
   "REG_Data".LCV300_Pologenie_ok := INT_TO_REAL("REG_Data".LCV300_Pologenie) / 10;
   //
   IF "REG_Data".PCV300_Pologenie_ok > 98.5 THEN
       "REG_Data".PCV300_Pologenie_ok := 100.0;
   END_IF;
   IF "REG_Data".LCV300_Pologenie_ok > 98.5 THEN
       "REG_Data".LCV300_Pologenie_ok := 100.0;
   END_IF;


   // Определение аварий и предупреждений для отображения на HMI
   // PCV300
   IF "REG_Data".PCV300_Message.Error OR "REG_Data".PCV300_Message.Term_error OR
       "REG_Data".PCV300_Message.Phase_failure OR "REG_Data".PCV300_Status.Error OR
       "REG_Data".PCV300_Status.Fail OR "REG_Master".PCV300_error
   THEN
       "Regs".PCV300_Alarm := true;
   ELSE
       "Regs".PCV300_Alarm := false;
   END_IF;

   IF "REG_Data".PCV300_Message.Warning OR "REG_Data".PCV300_Status.Warning
   THEN
       "Regs".PCV300_Warning := true;
   ELSE
       "Regs".PCV300_Warning := false;
   END_IF;

   // LCV300
   IF "REG_Data".LCV300_Message.Error OR "REG_Data".LCV300_Message.Term_error OR
       "REG_Data".LCV300_Message.Phase_failure OR "REG_Data".LCV300_Status.Error OR
       "REG_Data".LCV300_Status.Fail OR "REG_Master".LCV300_error
   THEN
       "Regs".LCV300_Alarm := true;
   ELSE
       "Regs".LCV300_Alarm := false;
   END_IF;

   IF "REG_Data".LCV300_Message.Warning OR "REG_Data".LCV300_Status.Warning
   THEN
       "Regs".LCV300_Warning := true;
   ELSE
       "Regs".LCV300_Warning := false;
   END_IF;

   // Для тестирования
   IF "REG_Master".LCV300_error THEN
       "REG_Master".test1 := "REG_Master".test1 + 1;
   END_IF;
END_FUNCTION

FUNCTION "Modbus_init" : Void   // FC11, SCL
{ S7_Optimized_Access := 'TRUE' }
VERSION : 0.1
BEGIN
   //************************************************ Регуляторы *****************************************************************
   "PortSettings".Regs."Port" := 258;
   "PortSettings".Regs.Baud := 19200;
   "PortSettings".Regs.Parity := 0;
   "REG_Master".Settings.MB_Addr := 1;
   "REG_Master".State := 10;

   "REG_Master".reqREGmaster := 0;
   "Modbus_Comm_Load_Regs".MODE := 4; // Operating mode 4 = Half duplex (RS485) two-wire mode
   "Modbus_Comm_Load_Regs"(REQ := true,
                           "PORT" := "PortSettings".Regs."Port",
                           BAUD := "PortSettings".Regs.Baud,
                           PARITY := "PortSettings".Regs.Parity,
                           FLOW_CTRL := 0,
                           RTS_ON_DLY := 0,
                           RTS_OFF_DLY := 0,
                           RESP_TO := 1000,
                           DONE => "PortSettings".Regs.Done,
                           ERROR => "PortSettings".Regs.Error,
                           STATUS => "PortSettings".Regs.Status,
                           MB_DB := "Modbus_Master_Regs".MB_DB);

   //************************************************ Передача на верхний уровень **************************************************
   "PortSettings".Up."Port" := 257;
   "PortSettings".Up.Baud := 9600;
   "PortSettings".Up.Parity := 0;

   "Modbus_Comm_Load_Up".MODE := 4; // Operating mode 4 = Half duplex (RS485) two-wire mode
   "Modbus_Comm_Load_Up"(REQ := true,
                         "PORT" := "PortSettings".Up."Port",
                         BAUD := "PortSettings".Up.Baud,
                         PARITY := "PortSettings".Up.Parity,
                         FLOW_CTRL := 0,
                         RTS_ON_DLY := 0,
                         RTS_OFF_DLY := 0,
                         RESP_TO := 1000,
                         DONE => "PortSettings".Up.Done,
                         ERROR => "PortSettings".Up.Error,
                         STATUS => "PortSettings".Up.Status,
                         MB_DB := "Modbus_Slave_Up".MB_DB);

   //************************************************ УВП **************************************************
   "MB_CLIENT_UVP".MB_Unit_ID := 1;
   "MB_CLIENT_UVP".MB_Transaction_ID := 1;
   "UVP_States".Connect_UVP.InterfaceId := 64;
   "UVP_States".Connect_UVP.ID := 1;
   "UVP_States".Connect_UVP.ActiveEstablished := true;
   "UVP_States".Connect_UVP.RemoteAddress.ADDR[1] := 10;
   "UVP_States".Connect_UVP.RemoteAddress.ADDR[2] := 158;
   "UVP_States".Connect_UVP.RemoteAddress.ADDR[3] := 144;
   "UVP_States".Connect_UVP.RemoteAddress.ADDR[4] := 30;
   "UVP_States".Connect_UVP.RemotePort := 502;
END_FUNCTION

FUNCTION "DATA_FC" : Void   // FC14, SCL
{ S7_Optimized_Access := 'TRUE' }
VERSION : 0.1
BEGIN
   // Перекладка данных в DATA

    "DATA".Measuring.PT100_Value := "PT100".Signal_AI.Value;
    "DATA".Measuring.PT100_Circuit := "PT100".Signal_AI.Circuit;
    "DATA".Measuring.TT100_Value := "TT100".Signal_AI.Value;
    "DATA".Measuring.TT100_Circuit := "TT100".Signal_AI.Circuit;
    "DATA".Measuring.LT100_Value := "LT100".Signal_AI.Value;
    "DATA".Measuring.LT100_Circuit := "LT100".Signal_AI.Circuit;
    "DATA".Measuring.AG100_Value := "AG100".Signal_AI.Value;
    "DATA".Measuring. AG100_Circuit := "AG100".Signal_AI.Circuit;
    "DATA".Measuring.PT200_Value := "PT200".Signal_AI.Value;
    "DATA".Measuring.PT200_Circuit := "PT200".Signal_AI.Circuit;
    "DATA".Measuring.TT200_Value := "TT200".Signal_AI.Value;
    "DATA".Measuring.TT200_Circuit := "TT200".Signal_AI.Circuit;
    "DATA".Measuring.LT200_Value := "LT200".Signal_AI.Value;
    "DATA".Measuring.LT200_Circuit := "LT200".Signal_AI.Circuit;
    "DATA".Measuring.AG200_Value := "AG200".Signal_AI.Value;
    "DATA".Measuring.AG200_Circuit := "AG200".Signal_AI.Circuit;
    "DATA".Measuring.TT500_Value := "TT500".Signal_AI.Value;
    "DATA".Measuring.TT500_Circuit := "TT500".Signal_AI.Circuit;
    "DATA".Measuring.PCV300_Pologenie := "REG_Data".PCV300_Pologenie_ok;
    "DATA".Measuring.LCV300_Pologenie := "REG_Data".LCV300_Pologenie_ok;
    //
    "DATA".Measuring.SIKG_Press := "UVP_Data".UVP1_Current_L1.UVP_Press;
    "DATA".Measuring.SIKG_Temp := "UVP_Data".UVP1_Current_L1.UVP_Temp;
    "DATA".Measuring.SIKG_Flow_ru := "UVP_Data".UVP1_Current_L1.UVP_vol_flow_work;
    "DATA".Measuring.SIKG_Flow_stu := "UVP_Data".UVP1_Current_L1.UVP_vol_flow_norm;
    "DATA".Measuring.SIKG_Flow_ru_prev2h := "UVP_Data".UVP1_Cumulative_L1.UVP_Vol_work_prev2h;
    "DATA".Measuring.SIKG_Flow_stu_prev2h := "UVP_Data".UVP1_Cumulative_L1.UVP_Vol_norm_prev2h;
    "DATA".Measuring.SIKG_Flow_ru_prevDay := "UVP_Data".UVP1_Cumulative_L1.UVP_Vol_work_prevDay;
    "DATA".Measuring.SIKG_Flow_stu_prevDay := "UVP_Data".UVP1_Cumulative_L1.UVP_Vol_norm_prevDay;
    "DATA".Measuring.SIKG_total := "UVP_Data".UVP1_Current_L1.UVP_Vol_norm;
    //
    "DATA".Measuring.SIKN_MassFlow := "UVP_Data".UVP1_Current_L2.UVP_vol_flow_work;
    "DATA".Measuring.SIKN_MassFlow_prev2h := "UVP_Data".UVP1_Cumulative_L2.UVP_Vol_work_prev2h;
    "DATA".Measuring.SIKN_MassFlow_prevDay := "UVP_Data".UVP1_Cumulative_L2.UVP_Vol_work_prevDay;
    "DATA".Measuring.SIKN_total := "UVP_Data".UVP1_Current_L2.UVP_Vol_work;

    // ***************************** СТАТУСЫ УСТРОЙСТВ *********************************
    // Статус XV100
    IF ("DI3".Slot.Pins[6] OR "DATA".Measuring.XV100_no_cmd_close OR "DATA".Measuring.XV100_no_cmd_open) THEN
        "DATA".Measuring.XV100_State := 3; // Авария
    ELSIF ("DI3".Slot.Pins[4] AND NOT "DI3".Slot.Pins[5]) THEN
        "DATA".Measuring.XV100_State := 2; // Открыт
    ELSIF ("DI3".Slot.Pins[5] AND NOT "DI3".Slot.Pins[4]) THEN
        "DATA".Measuring.XV100_State := 1; // Закрыт
    ELSE
        "DATA".Measuring.XV100_State := 0; // Неопределено
    END_IF;

    // Статус обогрева
    IF ("Head".Device.Fail > 0) THEN
        "DATA".Measuring.Head_State := 2; // Авария
    ELSIF ("Head".Device.State = 1) THEN
        "DATA".Measuring.Head_State := 1; // Включен
    ELSIF ("Head".Device.State = 0) THEN
        "DATA".Measuring.Head_State := 0; // Выключен
    END_IF;

    // Статус питания установки
    IF ("Power".Device.Fail > 0) THEN
        "DATA".Measuring.Power_State := 2; // Авария
    ELSIF ("Power".Device.State = 1) THEN
        "DATA".Measuring.Power_State := 1; // Включен
    ELSIF ("Power".Device.State = 0) THEN
        "DATA".Measuring.Power_State := 0; // Выключен
    END_IF;

    "DATA".Measuring.PCV300_Alarm := "Regs".PCV300_Alarm;
    "DATA".Measuring.PCV300_Warning := "Regs".PCV300_Warning;
    "DATA".Measuring.PCV300_Midle := "Regs".PCV300_Midle;
    "DATA".Measuring.PCV300_DIST := "REG_Data".PCV300_Message.Selector_DIST;
    "DATA".Measuring.PCV300_LOCAL := "REG_Data".PCV300_Message.Selector_LOCAL;
    "DATA".Measuring.LCV300_Alarm := "Regs".LCV300_Alarm;
    "DATA".Measuring.LCV300_Warning := "Regs".LCV300_Warning;
    "DATA".Measuring.LCV300_Midle := "Regs".LCV300_Midle;
    "DATA".Measuring.LCV300_DIST := "REG_Data".LCV300_Message.Selector_DIST;
    "DATA".Measuring.LCV300_LOCAL := "REG_Data".LCV300_Message.Selector_LOCAL;
    "DATA".Measuring.LS100 := "DI1".Slot.Pins[0];
    "DATA".Measuring.LS101 := "DI1".Slot.Pins[2];
    "DATA".Measuring.LS200 := "DI1".Slot.Pins[4];
    "DATA".Measuring.LS201 := "DI1".Slot.Pins[6];
    "DATA".Measuring.HS600_Emer_stop := "DI2".Slot.Pins[3];
    "DATA".Measuring.Head_run := "DI2".Slot.Pins[7];
    "DATA".Measuring.Power_run := "DI2".Slot.Pins[6];
    "DATA".Measuring.XV100_open := "DI3".Slot.Pins[4];
    "DATA".Measuring.XV100_close := "DI3".Slot.Pins[5];
    "DATA".Measuring.XV100_fault := "DI3".Slot.Pins[6];
    "DATA".Measuring.Spark := "DO1".Slot.Pins[4];

    "DATA".Measuring.PT100_HH_Alarm := "PT100".Signal_AI.HH_Alarm;
    "DATA".Measuring.PT100_H_Alarm := "PT100".Signal_AI.H_Alarm;
    "DATA".Measuring.PT100_L_Alarm := "PT100".Signal_AI.L_Alarm;
    "DATA".Measuring.PT100_LL_Alarm := "PT100".Signal_AI.LL_Alarm;
    "DATA".Measuring.PT100_Chan_Fail := "PT100".Signal_AI.Chan_Fail;
    "DATA".Measuring.PT100_Sim := "PT100".Signal_AI.Sim_En;

    "DATA".Measuring.TT100_HH_Alarm := "TT100".Signal_AI.HH_Alarm;
    "DATA".Measuring.TT100_H_Alarm := "TT100".Signal_AI.H_Alarm;
    "DATA".Measuring.TT100_L_Alarm := "TT100".Signal_AI.L_Alarm;
    "DATA".Measuring.TT100_LL_Alarm := "TT100".Signal_AI.LL_Alarm;
    "DATA".Measuring.TT100_Chan_Fail := "TT100".Signal_AI.Chan_Fail;
    "DATA".Measuring.TT100_Sim := "TT100".Signal_AI.Sim_En;

    "DATA".Measuring.LT100_HH_Alarm := "LT100".Signal_AI.HH_Alarm;
    "DATA".Measuring.LT100_H_Alarm := "LT100".Signal_AI.H_Alarm;
    "DATA".Measuring.LT100_L_Alarm := "LT100".Signal_AI.L_Alarm;
    "DATA".Measuring.LT100_LL_Alarm := "LT100".Signal_AI.LL_Alarm;
    "DATA".Measuring.LT100_Chan_Fail := "LT100".Signal_AI.Chan_Fail;
    "DATA".Measuring.LT100_Sim := "LT100".Signal_AI.Sim_En;

    "DATA".Measuring.AG100_HH_Alarm := "AG100".Signal_AI.HH_Alarm;
    "DATA".Measuring.AG100_H_Alarm := "AG100".Signal_AI.H_Alarm;
    "DATA".Measuring.AG100_L_Alarm := "AG100".Signal_AI.L_Alarm;
    "DATA".Measuring.AG100_LL_Alarm := "AG100".Signal_AI.LL_Alarm;
    "DATA".Measuring.AG100_Chan_Fail := "AG100".Signal_AI.Chan_Fail;
    "DATA".Measuring.AG100_Sim := "AG100".Signal_AI.Sim_En;

    "DATA".Measuring.PT200_HH_Alarm := "PT200".Signal_AI.HH_Alarm;
    "DATA".Measuring.PT200_H_Alarm := "PT200".Signal_AI.H_Alarm;
    "DATA".Measuring.PT200_L_Alarm := "PT200".Signal_AI.L_Alarm;
    "DATA".Measuring.PT200_LL_Alarm := "PT200".Signal_AI.LL_Alarm;
    "DATA".Measuring.PT200_Chan_Fail := "PT200".Signal_AI.Chan_Fail;
    "DATA".Measuring.PT200_Sim := "PT200".Signal_AI.Sim_En;

    "DATA".Measuring.TT200_HH_Alarm := "TT200".Signal_AI.HH_Alarm;
    "DATA".Measuring.TT200_H_Alarm := "TT200".Signal_AI.H_Alarm;
    "DATA".Measuring.TT200_L_Alarm := "TT200".Signal_AI.L_Alarm;
    "DATA".Measuring.TT200_LL_Alarm := "TT200".Signal_AI.LL_Alarm;
    "DATA".Measuring.TT200_Chan_Fail := "TT200".Signal_AI.Chan_Fail;
    "DATA".Measuring.TT200_Sim := "TT200".Signal_AI.Sim_En;

    "DATA".Measuring.LT200_HH_Alarm := "LT200".Signal_AI.HH_Alarm;
    "DATA".Measuring.LT200_H_Alarm := "LT200".Signal_AI.H_Alarm;
    "DATA".Measuring.LT200_L_Alarm := "LT200".Signal_AI.L_Alarm;
    "DATA".Measuring.LT200_LL_Alarm := "LT200".Signal_AI.LL_Alarm;
    "DATA".Measuring.LT200_Chan_Fail := "LT200".Signal_AI.Chan_Fail;
    "DATA".Measuring.LT200_Sim := "LT200".Signal_AI.Sim_En;

    "DATA".Measuring.AG200_HH_Alarm := "AG200".Signal_AI.HH_Alarm;
    "DATA".Measuring.AG200_H_Alarm := "AG200".Signal_AI.H_Alarm;
    "DATA".Measuring.AG200_L_Alarm := "AG200".Signal_AI.L_Alarm;
    "DATA".Measuring.AG200_LL_Alarm := "AG200".Signal_AI.LL_Alarm;
    "DATA".Measuring.AG200_Chan_Fail := "AG200".Signal_AI.Chan_Fail;
    "DATA".Measuring.AG200_Sim := "AG200".Signal_AI.Sim_En;

    "DATA".Measuring.TT500_HH_Alarm := "TT500".Signal_AI.HH_Alarm;
    "DATA".Measuring.TT500_H_Alarm := "TT500".Signal_AI.H_Alarm;
    "DATA".Measuring.TT500_L_Alarm := "TT500".Signal_AI.L_Alarm;
    "DATA".Measuring.TT500_LL_Alarm := "TT500".Signal_AI.LL_Alarm;
    "DATA".Measuring.TT500_Chan_Fail := "TT500".Signal_AI.Chan_Fail;
    "DATA".Measuring.TT500_Sim := "TT500".Signal_AI.Sim_En;



   // Запись команд из DATA
    "PT100".Signal_AI.Scal_Max_Eu := "DATA".Commands.PT100_Scal_Max_Eu;
    "PT100".Signal_AI.Scal_Min_Eu := "DATA".Commands.PT100_Scal_Min_Eu;
    "PT100".Signal_AI.HH_Lim := "DATA".Commands.PT100_HH_Lim;
    "PT100".Signal_AI.H_Lim := "DATA".Commands.PT100_H_Lim;
    "PT100".Signal_AI.L_Lim := "DATA".Commands.PT100_L_Lim;
    "PT100".Signal_AI.LL_Lim := "DATA".Commands.PT100_LL_Lim;
    "PT100".Signal_AI.Sim_Value := "DATA".Commands.PT100_Sim_Value;

    "TT100".Signal_AI.Scal_Max_Eu := "DATA".Commands.TT100_Scal_Max_Eu;
    "TT100".Signal_AI.Scal_Min_Eu := "DATA".Commands.TT100_Scal_Min_Eu;
    "TT100".Signal_AI.HH_Lim := "DATA".Commands.TT100_HH_Lim;
    "TT100".Signal_AI.H_Lim := "DATA".Commands.TT100_H_Lim;
    "TT100".Signal_AI.L_Lim := "DATA".Commands.TT100_L_Lim;
    "TT100".Signal_AI.LL_Lim := "DATA".Commands.TT100_LL_Lim;
    "TT100".Signal_AI.Sim_Value := "DATA".Commands.TT100_Sim_Value;

    "LT100".Signal_AI.Scal_Max_Eu := "DATA".Commands.LT100_Scal_Max_Eu;
    "LT100".Signal_AI.Scal_Min_Eu := "DATA".Commands.LT100_Scal_Min_Eu;
    "LT100".Signal_AI.HH_Lim := "DATA".Commands.LT100_HH_Lim;
    "LT100".Signal_AI.H_Lim := "DATA".Commands.LT100_H_Lim;
    "LT100".Signal_AI.L_Lim := "DATA".Commands.LT100_L_Lim;
    "LT100".Signal_AI.LL_Lim := "DATA".Commands.LT100_LL_Lim;
    "LT100".Signal_AI.Sim_Value := "DATA".Commands.LT100_Sim_Value;

    "AG100".Signal_AI.Scal_Max_Eu := "DATA".Commands.AG100_Scal_Max_Eu;
    "AG100".Signal_AI.Scal_Min_Eu := "DATA".Commands.AG100_Scal_Min_Eu;
    "AG100".Signal_AI.HH_Lim := "DATA".Commands.AG100_HH_Lim;
    "AG100".Signal_AI.H_Lim := "DATA".Commands.AG100_H_Lim;
    "AG100".Signal_AI.L_Lim := "DATA".Commands.AG100_L_Lim;
    "AG100".Signal_AI.LL_Lim := "DATA".Commands.AG100_LL_Lim;
    "AG100".Signal_AI.Sim_Value := "DATA".Commands.AG100_Sim_Value;

    "PT200".Signal_AI.Scal_Max_Eu := "DATA".Commands.PT200_Scal_Max_Eu;
    "PT200".Signal_AI.Scal_Min_Eu := "DATA".Commands.PT200_Scal_Min_Eu;
    "PT200".Signal_AI.HH_Lim := "DATA".Commands.PT200_HH_Lim;
    "PT200".Signal_AI.H_Lim := "DATA".Commands.PT200_H_Lim;
    "PT200".Signal_AI.L_Lim := "DATA".Commands.PT200_L_Lim;
    "PT200".Signal_AI.LL_Lim := "DATA".Commands.PT200_LL_Lim;
    "PT200".Signal_AI.Sim_Value := "DATA".Commands.PT200_Sim_Value;

    "TT200".Signal_AI.Scal_Max_Eu := "DATA".Commands.TT200_Scal_Max_Eu;
    "TT200".Signal_AI.Scal_Min_Eu := "DATA".Commands.TT200_Scal_Min_Eu;
    "TT200".Signal_AI.HH_Lim := "DATA".Commands.TT200_HH_Lim;
    "TT200".Signal_AI.H_Lim := "DATA".Commands.TT200_H_Lim;
    "TT200".Signal_AI.L_Lim := "DATA".Commands.TT200_L_Lim;
    "TT200".Signal_AI.LL_Lim := "DATA".Commands.TT200_LL_Lim;
    "TT200".Signal_AI.Sim_Value := "DATA".Commands.TT200_Sim_Value;

    "LT200".Signal_AI.Scal_Max_Eu := "DATA".Commands.LT200_Scal_Max_Eu;
    "LT200".Signal_AI.Scal_Min_Eu := "DATA".Commands.LT200_Scal_Min_Eu;
    "LT200".Signal_AI.HH_Lim := "DATA".Commands.LT200_HH_Lim;
    "LT200".Signal_AI.H_Lim := "DATA".Commands.LT200_H_Lim;
    "LT200".Signal_AI.L_Lim := "DATA".Commands.LT200_L_Lim;
    "LT200".Signal_AI.LL_Lim := "DATA".Commands.LT200_LL_Lim;
    "LT200".Signal_AI.Sim_Value := "DATA".Commands.LT200_Sim_Value;

    "AG200".Signal_AI.Scal_Max_Eu := "DATA".Commands.AG200_Scal_Max_Eu;
    "AG200".Signal_AI.Scal_Min_Eu := "DATA".Commands.AG200_Scal_Min_Eu;
    "AG200".Signal_AI.HH_Lim := "DATA".Commands.AG200_HH_Lim;
    "AG200".Signal_AI.H_Lim := "DATA".Commands.AG200_H_Lim;
    "AG200".Signal_AI.L_Lim := "DATA".Commands.AG200_L_Lim;
    "AG200".Signal_AI.LL_Lim := "DATA".Commands.AG200_LL_Lim;
    "AG200".Signal_AI.Sim_Value := "DATA".Commands.AG200_Sim_Value;

    "TT500".Signal_AI.Scal_Max_Eu := "DATA".Commands.TT500_Scal_Max_Eu;
    "TT500".Signal_AI.Scal_Min_Eu := "DATA".Commands.TT500_Scal_Min_Eu;
    "TT500".Signal_AI.HH_Lim := "DATA".Commands.TT500_HH_Lim;
    "TT500".Signal_AI.H_Lim := "DATA".Commands.TT500_H_Lim;
    "TT500".Signal_AI.L_Lim := "DATA".Commands.TT500_L_Lim;
    "TT500".Signal_AI.LL_Lim := "DATA".Commands.TT500_LL_Lim;
    "TT500".Signal_AI.Sim_Value := "DATA".Commands.TT500_Sim_Value;

    "PCV300".Setpoint := "DATA".Commands.PCV300_Setpoint;
    "PCV300".ManualValue := "DATA".Commands.PCV300_ManualValue;
    "PCV300".Retain.CtrlParams.Gain := "DATA".Commands.PCV300_Gain;
    "PCV300".Retain.CtrlParams.Ti := "DATA".Commands.PCV300_Ti;
    "PCV300".Retain.CtrlParams.Td := "DATA".Commands.PCV300_Td;
    "PCV300".Retain.CtrlParams.TdFiltRatio := "DATA".Commands.PCV300_TdFiltRatio;
    "PCV300".Config.OutputUpperLimit := "DATA".Commands.PCV300_OutputUpperLimit;
    "PCV300".Config.OutputLowerLimit := "DATA".Commands.PCV300_OutputLowerLimit;

    "LCV300".Setpoint := "DATA".Commands. LCV300_Setpoint;
    "LCV300".ManualValue := "DATA".Commands. LCV300_ManualValue;
    "LCV300".Retain.CtrlParams.Gain := "DATA".Commands. LCV300_Gain;
    "LCV300".Retain.CtrlParams.Ti := "DATA".Commands. LCV300_Ti;
    "LCV300".Retain.CtrlParams.Td := "DATA".Commands. LCV300_Td;
    "LCV300".Retain.CtrlParams.TdFiltRatio := "DATA".Commands. LCV300_TdFiltRatio;
    "LCV300".Config.OutputUpperLimit := "DATA".Commands. LCV300_OutputUpperLimit;
    "LCV300".Config.OutputLowerLimit := "DATA".Commands. LCV300_OutputLowerLimit;

    "PT100".Signal_AI.HH_Alarm_En := "DATA".Commands.PT100_HH_Alarm_En;
    "PT100".Signal_AI.H_Alarm_En := "DATA".Commands.PT100_H_Alarm_En;
    "PT100".Signal_AI.L_Alarm_En := "DATA".Commands.PT100_L_Alarm_En;
    "PT100".Signal_AI.LL_Alarm_En := "DATA".Commands.PT100_LL_Alarm_En;
    "PT100".Signal_AI.Sim_En := "DATA".Commands.PT100_Sim_En;

    "TT100".Signal_AI.HH_Alarm_En := "DATA".Commands.TT100_HH_Alarm_En;
    "TT100".Signal_AI.H_Alarm_En := "DATA".Commands.TT100_H_Alarm_En;
    "TT100".Signal_AI.L_Alarm_En := "DATA".Commands.TT100_L_Alarm_En;
    "TT100".Signal_AI.LL_Alarm_En := "DATA".Commands.TT100_LL_Alarm_En;
    "TT100".Signal_AI.Sim_En := "DATA".Commands.TT100_Sim_En;

    "LT100".Signal_AI.HH_Alarm_En := "DATA".Commands.LT100_HH_Alarm_En;
    "LT100".Signal_AI.H_Alarm_En := "DATA".Commands.LT100_H_Alarm_En;
    "LT100".Signal_AI.L_Alarm_En := "DATA".Commands.LT100_L_Alarm_En;
    "LT100".Signal_AI.LL_Alarm_En := "DATA".Commands.LT100_LL_Alarm_En;
    "LT100".Signal_AI.Sim_En := "DATA".Commands.LT100_Sim_En;

    "AG100".Signal_AI.HH_Alarm_En := "DATA".Commands.AG100_HH_Alarm_En;
    "AG100".Signal_AI.H_Alarm_En := "DATA".Commands.AG100_H_Alarm_En;
    "AG100".Signal_AI.L_Alarm_En := "DATA".Commands.AG100_L_Alarm_En;
    "AG100".Signal_AI.LL_Alarm_En := "DATA".Commands.AG100_LL_Alarm_En;
    "AG100".Signal_AI.Sim_En := "DATA".Commands.AG100_Sim_En;

    "PT200".Signal_AI.HH_Alarm_En := "DATA".Commands.PT200_HH_Alarm_En;
    "PT200".Signal_AI.H_Alarm_En := "DATA".Commands.PT200_H_Alarm_En;
    "PT200".Signal_AI.L_Alarm_En := "DATA".Commands.PT200_L_Alarm_En;
    "PT200".Signal_AI.LL_Alarm_En := "DATA".Commands.PT200_LL_Alarm_En;
    "PT200".Signal_AI.Sim_En := "DATA".Commands.PT200_Sim_En;

    "TT200".Signal_AI.HH_Alarm_En := "DATA".Commands.TT200_HH_Alarm_En;
    "TT200".Signal_AI.H_Alarm_En := "DATA".Commands.TT200_H_Alarm_En;
    "TT200".Signal_AI.L_Alarm_En := "DATA".Commands.TT200_L_Alarm_En;
    "TT200".Signal_AI.LL_Alarm_En := "DATA".Commands.TT200_LL_Alarm_En;
    "TT200".Signal_AI.Sim_En := "DATA".Commands.TT200_Sim_En;

    "LT200".Signal_AI.HH_Alarm_En := "DATA".Commands.LT200_HH_Alarm_En;
    "LT200".Signal_AI.H_Alarm_En := "DATA".Commands.LT200_H_Alarm_En;
    "LT200".Signal_AI.L_Alarm_En := "DATA".Commands.LT200_L_Alarm_En;
    "LT200".Signal_AI.LL_Alarm_En := "DATA".Commands.LT200_LL_Alarm_En;
    "LT200".Signal_AI.Sim_En := "DATA".Commands.LT200_Sim_En;

    "AG200".Signal_AI.HH_Alarm_En := "DATA".Commands.AG200_HH_Alarm_En;
    "AG200".Signal_AI.H_Alarm_En := "DATA".Commands.AG200_H_Alarm_En;
    "AG200".Signal_AI.L_Alarm_En := "DATA".Commands.AG200_L_Alarm_En;
    "AG200".Signal_AI.LL_Alarm_En := "DATA".Commands.AG200_LL_Alarm_En;
    "AG200".Signal_AI.Sim_En := "DATA".Commands.AG200_Sim_En;

    "TT500".Signal_AI.HH_Alarm_En := "DATA".Commands.TT500_HH_Alarm_En;
    "TT500".Signal_AI.H_Alarm_En := "DATA".Commands.TT500_H_Alarm_En;
    "TT500".Signal_AI.L_Alarm_En := "DATA".Commands.TT500_L_Alarm_En;
    "TT500".Signal_AI.LL_Alarm_En := "DATA".Commands.TT500_LL_Alarm_En;
    "TT500".Signal_AI.Sim_En := "DATA".Commands.TT500_Sim_En;

    "PCV300".ManualEnable := "DATA".Commands.PCV300_ManualEnable;
    "LCV300".ManualEnable := "DATA".Commands.LCV300_ManualEnable;

    // Включение обогрева
    IF "DATA".Commands.Head_cmd_on AND NOT "Head_cmd_on_prev" THEN
        "Head".Device.Cmd_On := 4;
        "DATA".Commands.Head_cmd_on := false;
    END_IF;
    "Head_cmd_on_prev" := "DATA".Commands.Head_cmd_on;

    // Выключение обогрева
    IF "DATA".Commands.Head_cmd_off AND NOT "Head_cmd_off_prev" THEN
        "Head".Device.Cmd_Off := 4;
        "DATA".Commands.Head_cmd_off := false;
    END_IF;
    "Head_cmd_off_prev" := "DATA".Commands.Head_cmd_off;

    // Сброс ошибки обогрева
    IF "DATA".Commands.Head_cmd_reset AND NOT "Power_reset_prev" THEN
        "Head".Device.Cmd_Reset_Error := 4;
        "DATA".Commands.Head_cmd_reset := false;
    END_IF;
    "Head_reset_prev" := "DATA".Commands.Head_cmd_reset;

    // Включение питания
    IF "DATA".Commands.Power_cmd_on AND NOT "Power_cmd_on_prev" THEN
        "Power".Device.Cmd_On := 4;
        "DATA".Commands.Power_cmd_on := false;
    END_IF;
    "Power_cmd_on_prev" := "DATA".Commands.Power_cmd_on;

    // Выключение питания
    IF "DATA".Commands.Power_cmd_off AND NOT "Power_cmd_off_prev" THEN
        "Power".Device.Cmd_Off := 4;
        "DATA".Commands.Power_cmd_off := false;
    END_IF;
    "Power_cmd_off_prev" := "DATA".Commands.Power_cmd_off;

    // Сброс ошибки питания
    IF "DATA".Commands.Power_cmd_reset AND NOT "Power_reset_prev" THEN
        "Power".Device.Cmd_Reset_Error := 4;
        "DATA".Commands.Power_cmd_reset := false;
    END_IF;
    "Power_reset_prev" := "DATA".Commands.Power_cmd_reset;

    IF NOT "Modbus_Comm_Load_Up".DONE THEN
        "Modbus_Comm_Load_Up".MODE := 4; // Operating mode 4 = Half duplex (RS485) two-wire mode
        "Modbus_Comm_Load_Up"(REQ := true,
                              "PORT" := "PortSettings".Up."Port",
                              BAUD := "PortSettings".Up.Baud,
                              PARITY := "PortSettings".Up.Parity,
                              FLOW_CTRL := 0,
                              RTS_ON_DLY := 0,
                              RTS_OFF_DLY := 0,
                              RESP_TO := 1000,
                              DONE => "PortSettings".Up.Done,
                              ERROR => "PortSettings".Up.Error,
                              STATUS => "PortSettings".Up.Status,
                              MB_DB := "Modbus_Slave_Up".MB_DB);
    END_IF;
END_FUNCTION